Staubli VAL3: OnF7.pgx

program OnF7()
begin
  //保存
  libSave()
  bInit=false
  popUpMsg("保存完成!")
end
